ABB RAPID module: 0013EDCA

MODULE RsTempModule
    LOCAL CONST robtarget Post_0_2:=[[376.634806152,280.293089577,110.099075176],[0.007466413,0.652788102,-0.756730114,-0.034226901],[-1,0,-1,5],[113.307522839,9E+09,9E+09,9E+09,9E+09,9E+09]];
    LOCAL PERS tooldata Tip_holder_mechanism:=[TRUE,[[-0.077,-53.377,109.892],[0.024406608,0.003647592,0.594886456,-0.803430842]],[0.5,[0,1.6,65.9],[1,0,0,0],0,0,0]];
PROC RsTempPath()
        MoveL Post_0_2,v1000,z100,Tip_holder_mechanism\WObj:=wobj0;
ENDPROC

ENDMODULE
